FUNCTION_BLOCK FB_LamparaComputada_ST
VAR_INPUT
    ManiobrasTotales: UINT := 2;
END_VAR
VAR_OUTPUT
    ManiobrasPendientes: UINT;
END_VAR
VAR
    Contador: CTD := (CV := ManiobrasTotales);

    Lampara AT %Q*: BOOL;
    Pulsador AT %I*: BOOL;    
    PulsadorReinicio AT %I*: BOOL;    
END_VAR

Contador(
    CD := Pulsador,
    LOAD := PulsadorReinicio,
    PV := ManiobrasTotales,
    Q => Lampara,
    CV => ManiobrasPendientes
    );

END_FUNCTION_BLOCK

(* stored: Version 1.1.0.1, ProductVersion 3.1.4024.15
   POU FB_LamparaComputada_ST: Id {2c52e490-02c0-48e6-8c38-6edb0e27b45e}, SpecialFunc None *)
